// TIA Portal V18 export
DATA_BLOCK "delete"   // DB72
VERSION : 0.1
// stored: AutoNumber true, DBAccessibleFromOPCUA true, InstanceOfName artLimiter, InstanceOfType FB
"artLimiter"
   // VAR_INPUT
   //    AckEr : Bool;
   //    UseArtLimitw : Bool;
   //    artLimfwd : Real;
   //    artLimRev : Real;
   //    para_in : "typeMotPara";
   // END_VAR
   // VAR_OUTPUT
   //    para_Artlimits : "typeMotPara";
   //    ER_WS : WString;
   //    ER : Bool;
   // END_VAR
BEGIN
END_DATA_BLOCK
